// TIA Portal V18 export
DATA_BLOCK "LED_Behavior_DB"   // DB51
VERSION : 0.1
// stored: AutoNumber true, DBAccessibleFromOPCUA true, InstanceOfName LED_Behavior, InstanceOfType FB
"LED_Behavior"
   // VAR_INPUT
   //    RED : Bool;
   //    GREEN : Bool;
   //    RED_BLINK : Bool;
   //    GREEN_BLINK : Bool;
   //    RED_GREEN_BLINK : Bool;
   // END_VAR
   // VAR_OUTPUT
   //    LED_1_Output : Bool;
   //    LED_2_Output : Bool;
   // END_VAR
   // VAR
   //    Red_Blink_Output : Bool;
   //    Green_Blink_Output : Bool;
   //    "Red/Green_Blink_Output" : Bool;
   //    Red_Blink_M : Bool;
   //    Red_Blink_S : Bool;
   //    Green_Blink_M : Bool;
   //    Green_Blink_S : Bool;
   //    Reset_Red_Blink : Bool;
   //    Reset_Green_Blink : Bool;
   //    Reset_RED_GREEN_Blink : Bool;
   //    RG_Blink_M : Bool;
   //    RG_Blink_S : Bool;
   // END_VAR
BEGIN
END_DATA_BLOCK
